{attribute 'GeneratedUsingTerminal: EL6080-0000-0016'}
{attribute addProperty BoxType "EL6080-0000-0016"}
{attribute addProperty Id "StatusAT %I*ARRAY [0..1] OF USINT0"}
{attribute addProperty CRC "4015942696"}
{attribute addProperty Size "0"}
TYPE Status_EF5E6C28 EXTENDS InputBase_8311D824 :
STRUCT
	{attribute addProperty Name "Status"}
	Status AT %I* : ARRAY [0..1] OF USINT;
END_STRUCT
END_TYPE

(* stored: Version 1.2.0.0, ProductVersion 3.1.4024.11
   DUT Status_EF5E6C28: Id {51d849d6-c318-4cc5-b0e3-b4613a9c87f8} *)
